FUNCTION_BLOCK ExampleFlashingLamp_Inheritance EXTENDS CyclicInstance
VAR
	// these timers are required to implement the flashing lamp object
	tick : ton;
	tock : ton;
END_VAR

//... no code should go here.

METHOD CyclicCall
VAR_INPUT
END_VAR
tick(in:=NOT tock.Q,pt:=T#1S);
tock(in:=tick.Q,pt:=T#1S);
END_METHOD

PROPERTY PUBLIC Output : BOOL
GET
Output := tick.Q;
END_GET
END_PROPERTY

END_FUNCTION_BLOCK

(* stored: Version 1.1.0.1, ProductVersion 3.1.4024.11
   POU ExampleFlashingLamp_Inheritance: Id {22e8ed2e-da40-4d53-b200-714dafe673cb}, SpecialFunc None
   Method CyclicCall: Id {2b7266d3-6c00-4a56-9644-69a5f1d4e5ac}
   Property Output: Id {f763be9f-9d11-4bd9-b6ca-0ea041ebbee6}
   Get Get: Id {6917ad8c-fa6a-400f-a66d-de2a05f1f040} *)
